TYPE tsPartSequence :
STRUCT
	asSequenceData:ARRAY[0..gc_uiStationNum] OF tsSequence;(*module sequence *)
END_STRUCT
END_TYPE

(* stored: Version 1.1.0.1, ProductVersion 3.1.4024.9
   DUT tsPartSequence: Id {a209d107-eeff-4e91-98f6-01d225359873} *)
